// TIA Portal V19 export
FUNCTION_BLOCK "Block_2"   // FB1, FBD
TITLE = FB
{ S7_Optimized_Access := 'TRUE' }
// stored: MemoryReserve 100, SetENOAutomatically false
   VAR
      HF : Array[0..10] of Bool;
   END_VAR
BEGIN

REGION Network 1: network 1
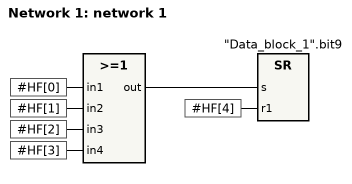
   IF #HF[0] OR #HF[1] OR #HF[2] OR #HF[3] THEN
       "Data_block_1".bit9 := TRUE;   // SR flip-flop
   END_IF;
   IF #HF[4] THEN "Data_block_1".bit9 := FALSE; END_IF;
END_REGION
END_FUNCTION_BLOCK
